/// This struct contains variables that
/// * are read from outside (e.g. HMI) to retrieve information about the unit's current state and (temporary) parameters (= `publish`) 
/// * are written from outside (e.g. HMI) to control the unit via ADS (= `subscribe`) 
TYPE PickerCom :
STRUCT
  Publish : PickerComPublish;
  Subscribe : PickerComSubscribe;
END_STRUCT
END_TYPE

(* stored: Version 1.1.0.1
   DUT PickerCom: Id {dc8d1297-514f-4114-b33d-b07f795c8ee1} *)
